PROGRAM QRob_StateMachine
VAR_INPUT
init_: BOOL:= FALSE;
//global aux state
G_STATE : INT := -1;
//comaper position to stop
Position : LREAL:= 0;
Velocity : REAL:=50;

END_VAR
VAR_OUTPUT
	State_complete : BOOL := FALSE;
	Act_Gl_State : INT := -1;
	Act_In_State : INT := -1;
	Act_Pos : REAL := -1;
END_VAR
VAR
	
//Axis status
Axis_state :BOOL:=FALSE;
	//internal aux state
I_STATE : INT:=-1;

//blocks to activate axis of qrob
Reset : MC_Reset;
ResetOut: ST_McOutputs;

PowerAxis1 : MC_Power;
/// debug function block output data 
PowerAxis1Out: ST_McOutputs;

MC_Stop: MC_Stop;

//blocks to move axis 
MoveAbsAxis1 :MC_MoveAbsolute;
MoveAbsoluteOut1: ST_McOutputs;

MC_MoveVelocity : MC_MoveVelocity;

//blocks to read paraemtres
MC_ReadActualPosition: MC_ReadActualPosition;



END_VAR

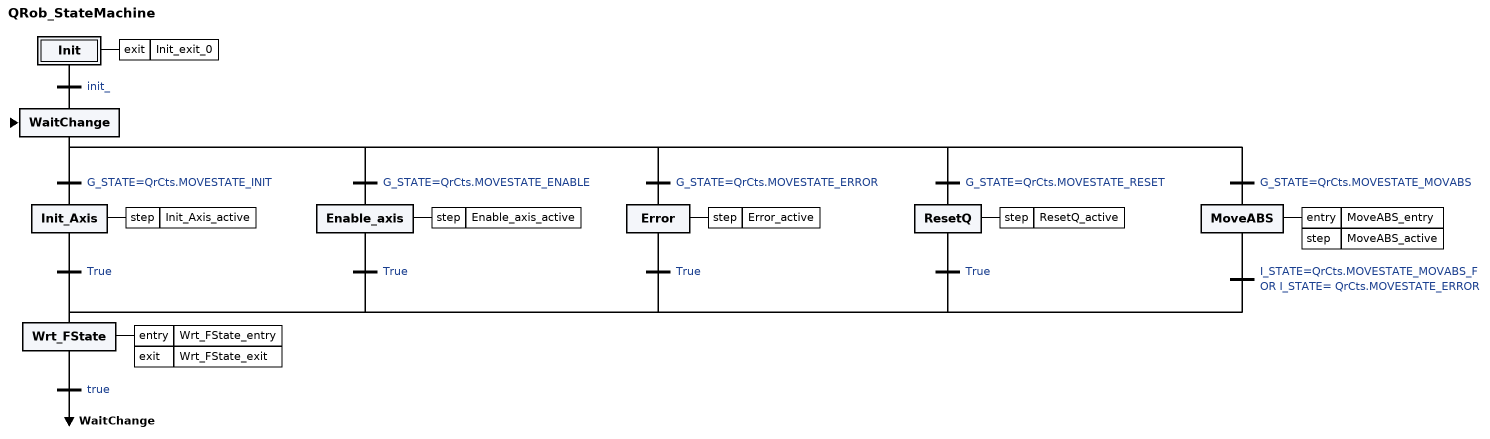
INITIAL_STEP Init:
    Init_exit_0(P0);  // exit action
END_STEP
TRANSITION FROM Init TO WaitChange
    := init_;
END_TRANSITION
STEP WaitChange:
END_STEP
TRANSITION FROM WaitChange TO Init_Axis
    := G_STATE=QrCts.MOVESTATE_INIT;
END_TRANSITION
STEP Init_Axis:
    Init_Axis_active(N);  // step action
END_STEP
TRANSITION FROM Init_Axis TO Wrt_FState
    := True;
END_TRANSITION
TRANSITION FROM WaitChange TO Enable_axis
    := G_STATE=QrCts.MOVESTATE_ENABLE;
END_TRANSITION
STEP Enable_axis:
    Enable_axis_active(N);  // step action
END_STEP
TRANSITION FROM Enable_axis TO Wrt_FState
    := True;
END_TRANSITION
TRANSITION FROM WaitChange TO Error
    := G_STATE=QrCts.MOVESTATE_ERROR;
END_TRANSITION
STEP Error:
    Error_active(N);  // step action
END_STEP
TRANSITION FROM Error TO Wrt_FState
    := True;
END_TRANSITION
TRANSITION FROM WaitChange TO ResetQ
    := G_STATE=QrCts.MOVESTATE_RESET;
END_TRANSITION
STEP ResetQ:
    ResetQ_active(N);  // step action
END_STEP
TRANSITION FROM ResetQ TO Wrt_FState
    := True;
END_TRANSITION
TRANSITION FROM WaitChange TO MoveABS
    := G_STATE=QrCts.MOVESTATE_MOVABS;
END_TRANSITION
STEP MoveABS:
    MoveABS_entry(P1);  // entry action
    MoveABS_active(N);  // step action
END_STEP
TRANSITION FROM MoveABS TO Wrt_FState
    := I_STATE=QrCts.MOVESTATE_MOVABS_F OR I_STATE= QrCts.MOVESTATE_ERROR;
END_TRANSITION
STEP Wrt_FState:
    Wrt_FState_entry(P1);  // entry action
    Wrt_FState_exit(P0);  // exit action
END_STEP
TRANSITION FROM Wrt_FState TO WaitChange
    := true;
END_TRANSITION

ACTION Act_MoveAbs:
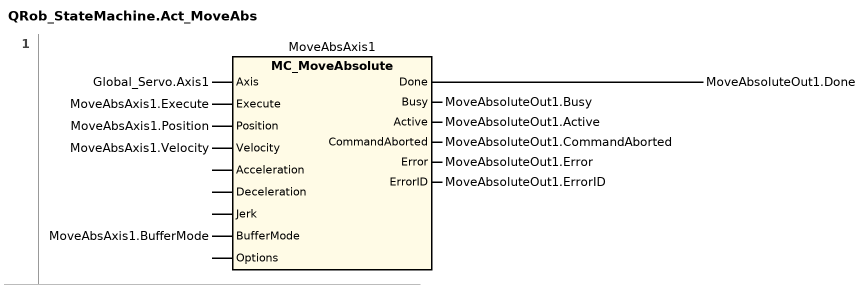
// NETWORK 1
MoveAbsAxis1(
    Axis := Global_Servo.Axis1,
    Execute := MoveAbsAxis1.Execute,
    Position := MoveAbsAxis1.Position,
    Velocity := MoveAbsAxis1.Velocity,
    BufferMode := MoveAbsAxis1.BufferMode,
    Busy => MoveAbsoluteOut1.Busy,
    Active => MoveAbsoluteOut1.Active,
    CommandAborted => MoveAbsoluteOut1.CommandAborted,
    Error => MoveAbsoluteOut1.Error,
    ErrorID => MoveAbsoluteOut1.ErrorID); // MC_MoveAbsolute
MoveAbsoluteOut1.Done := MoveAbsAxis1.Done;
END_ACTION

ACTION Act_Power:
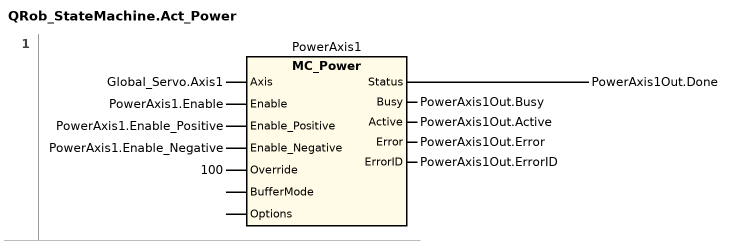
// NETWORK 1
PowerAxis1(
    Axis := Global_Servo.Axis1,
    Enable := PowerAxis1.Enable,
    Enable_Positive := PowerAxis1.Enable_Positive,
    Enable_Negative := PowerAxis1.Enable_Negative,
    Override := 100,
    Busy => PowerAxis1Out.Busy,
    Active => PowerAxis1Out.Active,
    Error => PowerAxis1Out.Error,
    ErrorID => PowerAxis1Out.ErrorID); // MC_Power
PowerAxis1Out.Done := PowerAxis1.Status;
END_ACTION

ACTION Act_Reset:
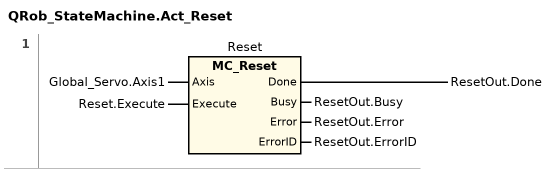
// NETWORK 1
Reset(
    Axis := Global_Servo.Axis1,
    Execute := Reset.Execute,
    Busy => ResetOut.Busy,
    Error => ResetOut.Error,
    ErrorID => ResetOut.ErrorID); // MC_Reset
ResetOut.Done := Reset.Done;
END_ACTION

ACTION Enable_axis_active:
//power on axis
PowerAxis1.Enable := TRUE;
PowerAxis1.Enable_Positive := TRUE;
PowerAxis1.Enable_Negative := TRUE;


IF PowerAxis1.Status THEN
	G_STATE := -1;
ELSIF PowerAxis1.Error THEN
	G_STATE := QrCts.MOVESTATE_ERROR;
END_IF

(* call the power function block *)
Act_Power();
Act_Reset();
Act_MoveAbs();
END_ACTION

ACTION Enable_axis_entry:
//power on axis
PowerAxis1.Enable := TRUE;
PowerAxis1.Enable_Positive := TRUE;
PowerAxis1.Enable_Negative := TRUE;
END_ACTION

ACTION Error_active:
IF Global_Servo.Axis1.Status.Error THEN
	G_STATE := QrCts.MOVESTATE_RESET;	(* axis error requires reset *)
ELSE
	G_STATE := QrCts.MOVESTATE_INIT;		(* function block errors don't need a reset *)
END_IF


(* call the power function block *)
Act_Power();
Act_Reset();
Act_MoveAbs();
END_ACTION

ACTION Init_Axis_active:
MoveAbsAxis1.Execute := FALSE;
Reset.Execute := FALSE;
G_State := QrCts.MOVESTATE_ENABLE;

(* call the power function block *)
Act_Power();
Act_Reset();
Act_MoveAbs();
END_ACTION

ACTION Init_Axis_entry:

END_ACTION

ACTION Init_Axis_exit:

END_ACTION

ACTION Init_exit:
// NETWORK 1
END_ACTION

ACTION Init_exit_0:
G_STATE:=QrCts.MOVESTATE_INIT;
END_ACTION

ACTION MoveABS_active:
IF MoveAbsAxis1.CommandAborted OR MoveAbsAxis1.Error THEN
	I_STATE := QrCts.MOVESTATE_ERROR;
ELSIF MoveAbsAxis1.Done THEN
	I_STATE := QrCts.MOVESTATE_MOVABS_F;
END_IF


//read internal variable and write over output variable
Act_In_State := I_STATE;


(* call the power function block *)
Act_Power();
Act_Reset();
Act_MoveAbs();
END_ACTION

ACTION MoveABS_entry:
MoveAbsAxis1.Position := Position;
MoveAbsAxis1.Velocity := Velocity;
MoveAbsAxis1.BufferMode := MC_Buffered;
MoveAbsAxis1.Execute := TRUE;

//write the retain state variable 
Act_Gl_State:=QrCts.MOVESTATE_MOVABS;
//read internal variable and write over output variable
I_STATE := QrCts.MOVESTATE_MOVABS_I;
Act_In_State := I_STATE;
END_ACTION

ACTION ResetQ_active:
Reset.Execute := TRUE;
IF Reset.Done THEN
	G_STATE := QrCts.MOVESTATE_INIT;
ELSIF Reset.Error THEN
	G_STATE := QrCts.MOVESTATE_INIT; (* can't do anything here *)
END_IF


(* call the power function block *)
Act_Power();
Act_Reset();
Act_MoveAbs();
END_ACTION

ACTION Wrt_FState_entry:
//write output variable to indicate that the robot execute the state 
State_complete := TRUE;
END_ACTION

ACTION Wrt_FState_exit:
//write output variable to indicate that the robot execute the state 
State_complete := FALSE;
init_:=FALSE;

G_STATE := -1;
//rest internat state variable
I_STATE :=-1;
END_ACTION

END_PROGRAM

(* stored: Version 1.1.0.1, ProductVersion 3.1.4024.4
   POU QRob_StateMachine: Id {dea1dd88-39fa-4c4e-93c5-ae49219992d0}, SpecialFunc None
   Action Act_MoveAbs: Id {6915af91-f4b1-4d40-99ec-2e82ddc50489}
   Action Act_Power: Id {85cbb579-2a28-41af-a636-5432fe4f3d32}
   Action Act_Reset: Id {72bd7d89-8767-4432-9292-a02562910a3e}
   Action Enable_axis_active: Id {726fecb4-69c6-4e7e-b391-d74d063e5215}
   Action Enable_axis_entry: Id {7c08845f-6242-4a60-abce-092305ddb52c}
   Action Error_active: Id {aa255cf8-ca48-4d1d-8627-2660654bd901}
   Action Init_Axis_active: Id {608179b8-0262-4a68-a08f-58e80770ad5d}
   Action Init_Axis_entry: Id {5fd46cfc-1bd1-434f-9105-dd6f5ba24956}
   Action Init_Axis_exit: Id {abd3e983-30fb-4cee-b74a-8a6f429417e0}
   Action Init_exit: Id {3e8dc8b2-5964-4b3d-b8a0-3598d1ff1d70}
   Action Init_exit_0: Id {ed758feb-5b02-4375-b9ea-b9b9faee0165}
   Action MoveABS_active: Id {bf482580-bca4-4945-86ee-79bf57cd951e}
   Action MoveABS_entry: Id {9d94e85e-c06d-4c66-9245-d026bb8c50a7}
   Action ResetQ_active: Id {c6601bd5-2819-48da-a47b-7c01580c8bc3}
   Action Wrt_FState_entry: Id {3fbfb66e-3783-4488-abed-6480d2af081b}
   Action Wrt_FState_exit: Id {e2a5e084-3023-4a1d-a625-641239d53d18} *)
